(*
  Base camera system with TcpIp communicatiom
  Implements callback function (rx_callback) for received TcpIp messages.   
*)
FUNCTION_BLOCK ABSTRACT FB_CameraTcpIp EXTENDS FB_CameraBase IMPLEMENTS I_TcpIp_RxMsgHandler

VAR
  sLastMessage              : STRING(GVL_TcpIp.TCP_RXDATA_SIZE);          (*rx telegram string*)
  nLastMessageSz            : UDINT;                                      (*receive message length *)
  sMemLastMessage           : STRING(GVL_TcpIp.TCP_RXDATA_SIZE);          (*mem rx telegram string*)
  nRxMsg                    : UDINT;                (*rx telegram counter*)
  bMsgReceived              : BOOL;                 (*we received a message*)
  sState                    : STRING;               (*state change event as string*)

  sLastErrorMessage         : STRING(GVL_TcpIp.TCP_RXDATA_SIZE);          (*rx telegram error string*)

  _pFbTcpIpClient           : POINTER TO FB_TcpClient;
END_VAR

METHOD ActivateCam : BOOL
VAR_INPUT
  iCameraSink : I_CameraSink;
END_VAR
ActivateCam := SUPER^.ActivateCam(iCameraSink:=iCameraSink);

IF _pFbTcpIpClient = 0 THEN
  LogError('No tcpip client assigned');
  ActivateCam := 0;
  RETURN;
END_IF

_pFbTcpIpClient^.bEnable := TRUE;
END_METHOD

PROPERTY bConnectionErr : BOOL
GET
IF _pFbTcpIpClient = 0 THEN RETURN; END_IF

IF _bActivated THEN
  IF NOT _pFbTcpIpClient^.bConnected OR _pFbTcpIpClient^.bError THEN
    bConnectionErr := TRUE;
  END_IF 
END_IF
END_GET
END_PROPERTY

METHOD CamTrigger
VAR_INPUT
  bOk             : BOOL;     // trigger is ok
	nPos            : DINT;     // camera triggered position
  nPosDeviation   : DINT;     // camera started deviation
END_VAR
SUPER^.CamTrigger(bOk:=bOk, nPos:=nPos, nPosDeviation:=nPosDeviation);
END_METHOD

METHOD DeactivateCam : BOOL
VAR_INPUT
  iSink : I_CameraSink;
END_VAR
DeactivateCam := SUPER^.DeactivateCam(iSink:=iSink);

IF _pFbTcpIpClient = 0 THEN
  LogError('No tcpip client assigned');
  DeactivateCam := 0;
  RETURN;
END_IF

_pFbTcpIpClient^.bEnable := FALSE;
END_METHOD

METHOD ABSTRACT GetCamStatus : BOOL
VAR_OUTPUT
  bConnectionOK  : BOOL;    // Camera connected
  bTeachOk       : BOOL;    // Teach successful
  nTeachedPoints : UDINT;   // Teached points for this job
  nScannedPoints : UDINT;   // Scanned points on current sheet
  bCamStarted    : BOOL;    // Camera trigger is active, cam started
  bCamDone       : BOOL;    // Camera finished on last CT
  bErrors        : ARRAY[1..GVL_Camera.nC_NbCamErrors] OF BOOL;  // generic error flag list
END_VAR
END_METHOD

METHOD rx_callback
VAR_INPUT
	sMessage	: CalmarCompTcpIp.ST_TcpMsg;
END_VAR
sLastMessage  := sMessage.sMessage;   // store message locally
nRxMsg        := nRxMsg + 1;
nLastMessageSz := LEN2(ADR(sLastMessage));

bMsgReceived  := TRUE;
END_METHOD

METHOD setTcpIpClient : BOOL
VAR_INPUT
  pTcpIpClient  : POINTER TO FB_TcpClient;
END_VAR
_pFbTcpIpClient := pTcpIpClient;
END_METHOD

METHOD state_callback
VAR_INPUT
	(* state change event as string (think to convert it to an enum for easier handling later)*)
	state	: STRING;
END_VAR
sState := state;   // store state locally
END_METHOD

END_FUNCTION_BLOCK

(* stored: Version 1.1.0.1, ProductVersion 3.1.4024.3
   POU FB_CameraTcpIp: Id {1219f4c9-29bb-471a-b078-b6b3aadb0883}, SpecialFunc None
   Method ActivateCam: Id {3ebd0870-e699-404f-9ba0-21ba4be68683}
   Property bConnectionErr: Id {4fda4592-4f45-4cbf-9cf8-5c0ac5d8d9fc}
   Get Get: Id {1c589870-4daf-48fb-8f17-987a6d156847}
   Method CamTrigger: Id {5faf1bcf-3bf4-4459-acb7-18b9546261f9}
   Method DeactivateCam: Id {d8fad887-f3ac-4c53-aaf7-eb439bc6a80e}
   Method GetCamStatus: Id {7e02114a-accf-46b9-bb54-3b92078e6773}
   Method rx_callback: Id {5f17216d-cbb6-44fc-9fc5-087403c2ab9d}
   Method setTcpIpClient: Id {c93f7529-e321-4200-beea-f3b2bb0e0db9}
   Method state_callback: Id {7e349b0b-5272-4a4a-80dd-0471e8328606} *)
